FUNCTION_BLOCK sdo_watch_time_logging IMPLEMENTS ITF_CoeSdoEventHandler
VAR_INPUT
END_VAR
VAR_OUTPUT
END_VAR
VAR
	cycle_time: ULINT;
	datetime_string: STRING;
	last_time :TIMESTRUCT;

END_VAR

PROPERTY lCycleTime : ULINT
GET
lCycleTime := cycle_time;
END_GET
END_PROPERTY

PROPERTY sDateTime : STRING
GET
sDateTime := datetime_string;
END_GET
END_PROPERTY

METHOD sdo_data_received : BOOL
VAR_INPUT
	command : REFERENCE TO CoeSdoCommand;
END_VAR
VAR
END_VAR

cycle_time := SYSTEMTIME_TO_FILETIME64(command.datetime) - SYSTEMTIME_TO_FILETIME64(last_time);
datetime_string := SYSTEMTIME_TO_ISO8601(
	systemTime := command.datetime,
	nBias := -540,
	bUTC := TRUE,
	nPrecision := 3
);
last_time := command.datetime;
END_METHOD

END_FUNCTION_BLOCK

(* stored: Version 1.1.0.1, ProductVersion 3.1.4024.12
   POU sdo_watch_time_logging: Id {9a93db3a-96b4-4a16-9fdd-1327b20ae3ba}, SpecialFunc None
   Property lCycleTime: Id {81d8446a-5a6d-415e-97c6-a9229c04ee7c}
   Get Get: Id {09886d6e-78b8-4621-825d-a58e2e6dfe48}
   Property sDateTime: Id {960fd723-2b23-4e02-b285-8652285c2da8}
   Get Get: Id {5668f501-4460-47e8-914a-57690e825ef1}
   Method sdo_data_received: Id {3cc0f1c8-17f0-44f9-aed7-dce818bc42b9} *)
